(*~
    <docu>
        <summary>
            TcoAxisExchangeDataTask task is a remote task  <see cref="PlcDocu.TcoCore.RemoteTask"/> with a paramater.
        </summary>
        <param name="_identifier">The Identifier, ID  of an entity on which a CRUD operation should be executed</param>
        <remarks>Inxton is required for this feature to work</remarks>
    </docu>
~*)
FUNCTION_BLOCK TcoAxisExchangeDataTask EXTENDS TcoCore.TcoRemoteTask
VAR
    (*~
    <docu>
        <summary>
            The Identifier, ID  of an entity on which a CRUD operation should be executed.
        </summary>
    </docu>
    ~*)
    _identifier : STRING(255);
    _doesNotExist : BOOL;
    _exchangeSuccessfuly : BOOL;
END_VAR

SUPER^();

PROPERTY PUBLIC DoesNotExist : bool
GET
DoesNotExist := _doesNotExist;
END_GET
END_PROPERTY

PROPERTY ReadSuccessfuly : bool
GET
ReadSuccessfuly := _exchangeSuccessfuly;
END_GET
END_PROPERTY

(*~
    <docu>
        <summary>
            Restores this instance to the Ready state. Can be called explicitly or from within one of the restore mechanisms.
            <para>
                See also <see cref="PlcDocu.TcoCore.TcoTask.AutoRestorable()"/>
            </para>
        </summary>
    </docu>
~*)
METHOD Restore : ITcoRestorable
VAR
END_VAR
_doesNotExist := FALSE;
//_identifier:='';
_exchangeSuccessfuly := FALSE;
SUPER^.Restore();
END_METHOD

METHOD WithId : REFERENCE TO TcoAxisExchangeDataTask
VAR_INPUT
    (*~
    <docu>
        <summary>
            The Identifier, ID  of an entity on which a CRUD operation should be executed.
        </summary>
    </docu>
    ~*)
    inIdentifier : STRING(254);
END_VAR
THIS^._identifier := inIdentifier;
WithId REF= THIS^;
THIS^.Messenger.Build().Append('<#Loading/saving data item with id:#> ').Append(_identifier).As().AsTrace();
END_METHOD

END_FUNCTION_BLOCK

(* stored: Version 1.1.0.1, ProductVersion 3.1.4024.12
   POU TcoAxisExchangeDataTask: Id {70b5fecb-d418-0a63-1b9f-b3b6f1baa87a}, SpecialFunc None
   Property DoesNotExist: Id {c79d3b2e-4221-0f94-1d2c-f58883eb0746}
   Get Get: Id {c8e4cee1-9159-0576-0009-d3984172f572}
   Property ReadSuccessfuly: Id {b5a186eb-e088-0f79-198b-a32de57d7878}
   Get Get: Id {22aa8aab-5593-06bd-0cf4-911d4b855aec}
   Method Restore: Id {c3411037-c1a6-0f43-1be4-9b3d98b2d53c}
   Method WithId: Id {7131bbd6-0b83-0114-15d0-afa3b79f5b85} *)
